// TIA Portal V17 export
// export: Created 2024-08-26T21:10:53.8431192Z, ExportSetting WithDefaults, DisplayName Totally Integrated Automation Portal, DisplayVersion V17 Update 7, DisplayName TIA Portal Openness, DisplayVersion V17 Update 7, DisplayName TIA Portal Version Control Interface, DisplayVersion V17, DisplayName SINAMICS Startdrive Advanced, DisplayVersion V17 SP2, DisplayName SINAMICS Startdrive G110M, G120, G120C, G120D, G120P, G115D, DisplayVersion V17 SP2, DisplayName SINAMICS Startdrive G130, G150, S120, S150, SINAMICS MV, S210, DisplayVersion V17 SP2, DisplayName STEP 7 Professional, DisplayVersion V17 Update 7, DisplayName STEP 7 Safety, DisplayVersion V17 Update 6, DisplayName WinCC Advanced / Unified PC, DisplayVersion V17 Update 7
VAR_GLOBAL   // PLC tag table "alarmMemory"
   alarm0 AT %MW100 : Int;   // alarm number
   alarm1 AT %MW102 : Int;   // alarm number
   alarm2 AT %MW104 : Int;
   retIolink AT %MW108 : Int;
   retManifold AT %MW112 : Int;
   retEuchner AT %MW106 : Int;
   retIolink2 AT %MW110 : Int;
   removeScannerError AT %MW6 : Word;
   Green AT %M2.0 : Bool;
   yellow AT %M2.1 : Bool;
   red AT %M2.2 : Bool;
   qRedTurretSolid AT %M3.6 : Bool;
   kkkk AT %M8.1 : Bool;
   hmifinalTorqueAngle AT %MW10 : Word;
END_VAR
